{attribute 'qualified_only'}
// ------------------------------------------------------------------------- 
//  SRCI Robot Library                                                
// ------------------------------------------------------------------------- 
//                                                                           
//  Object:      TriggerModeLimit                                       
//  Author:      Thorsten Brach                                                
//  Date:        2024-06-01
//
//  Description:                                              
//   
//                                                                           
//  Copyright: 
//    (C) 2024 Thorsten Brach. All rights reserved                                                                         
//                                                                           
//  Disclaimer:                                                                           
//    This project is provided without any guarantee and can be used for   
//    private and commercial purposes. Any commercial use is at the user’s 
//    own risk and responsibility.
//
// -------------------------------------------------------------------------
TYPE TriggerModeLimit :
(
	/// 0: Invalid (default)
  INVALID := 0,
  /// 1: Joint current in mA
  JOINT_CURRENT := 1,
  /// 2: Force in Nm
  FORCE := 2,
  /// 3: Following error. The distance of the robot position from the path that was calculated
  FOLLOWING_ERROR := 3,
  /// Temperature in °C
  TEMPERATURE := 4  
)SINT;
END_TYPE

{attribute 'qualified_only'}
// ------------------------------------------------------------------------- 
//  SRCI Robot Library                                                
// ------------------------------------------------------------------------- 
//                                                                           
//  Object:      TriggerModeMeasurement                                       
//  Author:      Thorsten Brach                                                
//  Date:        2024-06-01
//
//  Description:                                              
//   
//                                                                           
//  Copyright: 
//    (C) 2024 Thorsten Brach. All rights reserved                                                                         
//                                                                           
//  Disclaimer:                                                                           
//    This project is provided without any guarantee and can be used for   
//    private and commercial purposes. Any commercial use is at the user’s 
//    own risk and responsibility.
//
// -------------------------------------------------------------------------
TYPE TriggerModeMeasurement :
(
	/// (default) No trigger related behavior
  NO_TRIGGER := 0,
  /// 1: Starts the measurement with the positive trigger event and stops it with the negative trigger event 
  ///    when the trigger function with the identical EmitterID is activated.
  POSITIVE_START_NEGATIVE_STOP := 1,
  /// 2: Starts and stops the measurement with the positive trigger event 
  ///    when the trigger function with the identical EmitterID is activated.
  POSITIVE_START_STOP := 2
)USINT;
END_TYPE

{attribute 'qualified_only'}
// ------------------------------------------------------------------------- 
//  SRCI Robot Library                                                
// ------------------------------------------------------------------------- 
//                                                                           
//  Object:      TriggerReactionMode                                       
//  Author:      Thorsten Brach                                                
//  Date:        2024-06-01
//
//  Description:                                              
//   
//                                                                           
//  Copyright: 
//    (C) 2024 Thorsten Brach. All rights reserved                                                                         
//                                                                           
//  Disclaimer:                                                                           
//    This project is provided without any guarantee and can be used for   
//    private and commercial purposes. Any commercial use is at the user’s 
//    own risk and responsibility.
//
// -------------------------------------------------------------------------
TYPE TriggerReactionMode :
(
/// No reaction (default).
  NO_REACTION := 0,
  /// Interrupt: Robot movement is paused. Movement can be continued by function GroupContinue.
  INTERRUPT := 1,
  /// GroupStop: Robot stops the movement and brings all axes to a halt. Movements aborted by this command cannot be continued.
  GROUP_STOP := 2,
  /// Disable robot: The robot’s drives are disabled. This leads to the robot state "Not enabled" (see chapter 5.5.3).
  DISABLE_ROBOT := 3,
  /// Stop actual motion command: Robot movement is paused. Movement can be continued by the next motion command.
  STOP_ACTUAL_MOTION_COMMAND := 4
)SINT;
END_TYPE

{attribute 'qualified_only'}
// ------------------------------------------------------------------------- 
//  SRCI Robot Library                                                
// ------------------------------------------------------------------------- 
//                                                                           
//  Object:      TurnMode                                       
//  Author:      Thorsten Brach                                                
//  Date:        2024-06-01
//
//  Description:                                              
//   
//                                                                           
//  Copyright: 
//    (C) 2024 Thorsten Brach. All rights reserved                                                                         
//                                                                           
//  Disclaimer:                                                                           
//    This project is provided without any guarantee and can be used for   
//    private and commercial purposes. Any commercial use is at the user’s 
//    own risk and responsibility.
//
// -------------------------------------------------------------------------
TYPE TurnMode :
(
  /// Use TurnNumber in position
	USE_TURN_NUMBER := 0,
  ///  Do not change TurnNumber with this movement
  SAME            := 1,
  /// TurnNumber in position is not used but the Robot is free to change TurnNumber
  FREE            := 2
)USINT;
END_TYPE

{attribute 'qualified_only'}
// ------------------------------------------------------------------------- 
//  SRCI Robot Library                                                
// ------------------------------------------------------------------------- 
//                                                                           
//  Object:      WorkAreaReactionMode                                       
//  Author:      Thorsten Brach                                                
//  Date:        2024-06-01
//
//  Description:                                              
//   
//                                                                           
//  Copyright: 
//    (C) 2024 Thorsten Brach. All rights reserved                                                                         
//                                                                           
//  Disclaimer:                                                                           
//    This project is provided without any guarantee and can be used for   
//    private and commercial purposes. Any commercial use is at the user’s 
//    own risk and responsibility.
//
// -------------------------------------------------------------------------
TYPE WorkAreaReactionMode :
(
  /// 0: No reaction (default)
  /// • RC reports violation
  /// • Robot is not stopped
  NO_REACTION := 0,
  /// 
  /// 1: Abort
  /// • RC reports violation
  /// • RC returns error
  /// • Robot is stopped
  /// • Sequence buffer emptied
  ABORT := 1,
  /// 2: Interrupt
  /// • RC reports violation
  /// • Robot movement is paused
  /// • Movement can be continued by function GroupContinue
   INTERRUPT := 2
)USINT;
END_TYPE

{attribute 'qualified_only'}
// ------------------------------------------------------------------------- 
//  SRCI Robot Library                                                
// ------------------------------------------------------------------------- 
//                                                                           
//  Object:      ActiveCommandRegisterState                                       
//  Author:      Thorsten Brach                                                
//  Date:        2024-06-01
//
//  Description:                                              
//   
//                                                                           
//  Copyright: 
//    (C) 2024 Thorsten Brach. All rights reserved                                                                         
//                                                                           
//  Disclaimer:                                                                           
//    This project is provided without any guarantee and can be used for   
//    private and commercial purposes. Any commercial use is at the user’s 
//    own risk and responsibility.
//
// -------------------------------------------------------------------------
TYPE ActiveCommandRegisterState :
(
  /// IS_FREE denotes not used but available resources (empty slots in the ACR).
	IS_FREE        := 0,
  /// IS_PROCESSING CMDs are actively being processed by client or server. 
  /// In terms of CMD category, IS_PROCESSING also describes commands whose tasks are not currently being executed (not ACTIVE), 
  /// but e.g. a CMD waiting in the Sequence buffer.
  IS_PROCESSING := 1,
  /// IS_FINAL states are reached on CMD termination. Execution of this Task has been finished and its results can be examined.
  IS_FINAL    := 2
);
END_TYPE

{attribute 'qualified_only'}
// ------------------------------------------------------------------------- 
//  SRCI Robot Library                                                
// ------------------------------------------------------------------------- 
//                                                                           
//  Object:      BufferStateCmd                                       
//  Author:      Thorsten Brach                                                
//  Date:        2024-06-01
//
//  Description:                                              
//   
//                                                                           
//  Copyright: 
//    (C) 2024 Thorsten Brach. All rights reserved                                                                         
//                                                                           
//  Disclaimer:                                                                           
//    This project is provided without any guarantee and can be used for   
//    private and commercial purposes. Any commercial use is at the user’s 
//    own risk and responsibility.
//
// -------------------------------------------------------------------------
TYPE BufferStateCmd :
(
 // PDF Seite 353 
  EMPTY            := 0,
	CREATED          := 1,
  UPDATE_AVAILABLE := 2,
  SENDING          := 3,
  PROCESSED        := 4  
);
END_TYPE

{attribute 'qualified_only'}
// ------------------------------------------------------------------------- 
//  SRCI Robot Library                                                
// ------------------------------------------------------------------------- 
//                                                                           
//  Object:      BufferStateRsp                                       
//  Author:      Thorsten Brach                                                
//  Date:        2024-06-01
//
//  Description:                                              
//   
//                                                                           
//  Copyright: 
//    (C) 2024 Thorsten Brach. All rights reserved                                                                         
//                                                                           
//  Disclaimer:                                                                           
//    This project is provided without any guarantee and can be used for   
//    private and commercial purposes. Any commercial use is at the user’s 
//    own risk and responsibility.
//
// -------------------------------------------------------------------------
TYPE BufferStateRsp :
(
 // PDF Seite 353 
  EMPTY            := 0,
  RECEIVING        := 1,
  RECEIVED         := 2,
  PROCESSED        := 3  
);
END_TYPE

{attribute 'qualified_only'}
// ------------------------------------------------------------------------- 
//  SRCI Robot Library                                                
// ------------------------------------------------------------------------- 
//                                                                           
//  Object:      CmdMessageState                                       
//  Author:      Thorsten Brach                                                
//  Date:        2024-06-01
//
//  Description:                                              
//   
//                                                                           
//  Copyright: 
//    (C) 2024 Thorsten Brach. All rights reserved                                                                         
//                                                                           
//  Disclaimer:                                                                           
//    This project is provided without any guarantee and can be used for   
//    private and commercial purposes. Any commercial use is at the user’s 
//    own risk and responsibility.
//
// -------------------------------------------------------------------------
TYPE CmdMessageState :
(
  /// No operation or process is active
  EMPTY := 0,
  /// Created but not yet started
  CREATED := 1,
  /// Buffered and awaiting execution
  BUFFERED := 2,
  /// Buffered in planner for future execution
  BUFFERED_IN_PLANNER := 3,
  /// Currently active and in progress
  ACTIVE := 4,
  /// Interrupted and awaiting continuation
  INTERRUPTED := 5,
  /// Requested for abort
  ABORT_REQUEST := 6,
  /// Successfully completed
  DONE := 10,
  /// Aborted before completion
  ABORTED := 14,
  /// Encountered an error during execution
  ERROR := 15
)USINT;
END_TYPE

{attribute 'qualified_only'}
// ------------------------------------------------------------------------- 
//  SRCI Robot Library                                                
// ------------------------------------------------------------------------- 
//                                                                           
//  Object:      InitializationState                                       
//  Author:      Thorsten Brach                                                
//  Date:        2024-06-01
//
//  Description:                                              
//   
//                                                                           
//  Copyright: 
//    (C) 2024 Thorsten Brach. All rights reserved                                                                         
//                                                                           
//  Disclaimer:                                                                           
//    This project is provided without any guarantee and can be used for   
//    private and commercial purposes. Any commercial use is at the user’s 
//    own risk and responsibility.
//
// -------------------------------------------------------------------------
TYPE InitializationState :
(
  /// Default
  DEFAULT := 0,
  /// Error: Telegram control does not match the telegram state
  ERROR_TELEGRAM_CONTROL := 161,
  /// Error: Initialization lost for unknown reason. See message log after reinitializing
  ERROR_INIT_LOST := 162,
  /// Error: Telegram length does not match the length provided in the communication interface.
  ERROR_TELEGRAM_LENGTH := 163,
  /// Error: Incompatible major SRCI version
  ERROR_INCOMPATIBLE_SRCI := 164,
  /// Error: Lifesign timeout
  ERROR_LIFESIGN_TIMEOUT := 165,
  /// Error: The selected optional cyclic data does not fit in the given telegram size
  ERROR_CYCLIC_DATA_MISMATCH := 166,
  /// Error: The robot interface was reset after being initialized
  ERROR_INTERFACE_RESET := 167,
  /// Error: Telegram sequence timeout
  ERROR_SEQUENCE_TIMEOUT := 168,
  /// Error: The telegram number changed after initialization
  ERROR_TELEGRAM_NUMBER_CHANGED := 169,
  /// Error: Invalid AxesGroupID
  ERROR_INVALID_AXES_GROUP := 170,
  /// Error: Telegram number is invalid. E.g. TwoSequences is only activated in one direction
  ERROR_INVALID_TELEGRAM_NUMBER := 171,
  /// Error: Telegram Number is not supported
  ERROR_TELEGRAM_NUMBER_NOT_SUPPORTED := 172,
  /// Ready to resume: The RC is currently not initialized but has state in the ACR
  READY_TO_RESUME := 253,
  /// Ready for initialization: The RC is currently not initialized and has no state in the ACR
  READY_FOR_INITIALIZATION := 254,
  /// Initialized: The RC state is Initialized
  INITIALIZED := 255
);
END_TYPE

{attribute 'qualified_only'}
// ------------------------------------------------------------------------- 
//  SRCI Robot Library                                                
// ------------------------------------------------------------------------- 
//                                                                           
//  Object:      RaPowerState                                       
//  Author:      Thorsten Brach                                                
//  Date:        2024-06-01
//
//  Description:                                              
//   
//                                                                           
//  Copyright: 
//    (C) 2024 Thorsten Brach. All rights reserved                                                                         
//                                                                           
//  Disclaimer:                                                                           
//    This project is provided without any guarantee and can be used for   
//    private and commercial purposes. Any commercial use is at the user’s 
//    own risk and responsibility.
//
// -------------------------------------------------------------------------
TYPE RaPowerState :
(
  /// Robot drives disabled. Robot cannot be moved
	NOT_ENABLED := 0,
  /// Robot drives powered on. Robot can be moved according to sequence state
  ENABLED := 1
)USINT;
END_TYPE

{attribute 'qualified_only'}
// ------------------------------------------------------------------------- 
//  SRCI Robot Library                                                
// ------------------------------------------------------------------------- 
//                                                                           
//  Object:      RaSequenceState                                       
//  Author:      Thorsten Brach                                                
//  Date:        2024-06-01
//
//  Description:                                              
//   
//                                                                           
//  Copyright: 
//    (C) 2024 Thorsten Brach. All rights reserved                                                                         
//                                                                           
//  Disclaimer:                                                                           
//    This project is provided without any guarantee and can be used for   
//    private and commercial purposes. Any commercial use is at the user’s 
//    own risk and responsibility.
//
// -------------------------------------------------------------------------
TYPE RaSequenceState :
(
  /// Robot can be moved by incoming command
	IDLE := 0,
  /// RC is processing command in active sequence
  EXECUTING := 1,
  /// Interrupt is active. Robot is waiting for Continue
  INTERRUPTED := 2
)USINT;
END_TYPE

{attribute 'qualified_only'}
// ------------------------------------------------------------------------- 
//  SRCI Robot Library                                                
// ------------------------------------------------------------------------- 
//                                                                           
//  Object:      RiState                                       
//  Author:      Thorsten Brach                                                
//  Date:        2024-06-01
//
//  Description:                                              
//   
//                                                                           
//  Copyright: 
//    (C) 2024 Thorsten Brach. All rights reserved                                                                         
//                                                                           
//  Disclaimer:                                                                           
//    This project is provided without any guarantee and can be used for   
//    private and commercial purposes. Any commercial use is at the user’s 
//    own risk and responsibility.
//
// -------------------------------------------------------------------------
TYPE RiState :
(
  /// RI is not initialized
	NOT_INITIALIZED := 0,
  /// Initialization finished successfully
  INITIALIZED := 1,
  /// Data between RC and PLC has been synchronized
  SYNCHRONIZED := 2
)USINT;
END_TYPE

{attribute 'qualified_only'}
// ------------------------------------------------------------------------- 
//  SRCI Robot Library                                                
// ------------------------------------------------------------------------- 
//                                                                           
//  Object:      AreaType                                       
//  Author:      Thorsten Brach                                                
//  Date:        2024-06-01
//
//  Description:                                              
//   
//                                                                           
//  Copyright: 
//    (C) 2024 Thorsten Brach. All rights reserved                                                                         
//                                                                           
//  Disclaimer:                                                                           
//    This project is provided without any guarantee and can be used for   
//    private and commercial purposes. Any commercial use is at the user’s 
//    own risk and responsibility.
//
// -------------------------------------------------------------------------
TYPE AreaType :
(
  /// 0: Axes
	AXES := 0,
  /// 1: Box (default)
  BOX := 1,
  /// 2: Cylinder
  CYLINDER := 2,
  /// 3: Sphere (only DefinitionMode 1)
  SPHERE := 3
)USINT;
END_TYPE

{attribute 'qualified_only'}
// ------------------------------------------------------------------------- 
//  SRCI Robot Library                                                
// ------------------------------------------------------------------------- 
//                                                                           
//  Object:      AxesGroupParameterCmdEntries                                       
//  Author:      Thorsten Brach                                                
//  Date:        2024-06-01
//
//  Description:                                              
//   
//                                                                           
//  Copyright: 
//    (C) 2024 Thorsten Brach. All rights reserved                                                                         
//                                                                           
//  Disclaimer:                                                                           
//    This project is provided without any guarantee and can be used for   
//    private and commercial purposes. Any commercial use is at the user’s 
//    own risk and responsibility.
//
// -------------------------------------------------------------------------
TYPE AxesGroupParameterCmdEntries :
(
  /// Handles multiple mechanisms required for operation of the interface
  RobotTask := 0, // No function code  
  /// Read robot-specific data from the RC
  ReadRobotData := 9002,  
  /// Enable/Disable robot into RA power state "Enabled"
  EnableRobot := 1,  
  /// Acknowledgement all pending errors
  GroupReset := 2,  
  /// Read the actual position – TCP: X…RZ + config/Turn, Joint: (J1…E6)
  ReadActualPosition := 3,
  /// Read the actual position cyclically
  ReadActualPositionCyclic := 4,   
  /// Read D-H-parameters of robot
  ReadDHParameter := 5,  
  /// Restart/reboot of the RC
  RestartController := 6,  
  /// Read actual TCP velocity
  ReadActualTCPVelocity := 7,  
  /// Login on RC from PLC
  UserLogin := 8,  
  /// Switch language of robot teach pendant from PLC
  SwitchLanguage := 9,  
  /// Reads and writes specific configuration parameters on RC that are required for the RI to work
  ExchangeConfiguration := 10,  
  /// Set active sequence
  SetSequence := 11,  
  /// Change actual speed override
  ChangeSpeedOverride := 12,  
  /// Read error codes of pending errors and move them into user data block "RobotData"
  ReadMessages := 13,  
  /// Read reference values of robot dynamics for path movement
  ReadRobotReferenceDynamics := 14,  
  /// Change configuration of selected user frame number
  WriteFrameData := 15,  
  /// Change configuration of selected tool number
  WriteToolData := 16,  
  /// Change configuration of selected payload number
  WriteLoadData := 17,  
  /// Write reference values of robot dynamics for path movement
  WriteRobotReferenceDynamics := 18,  
  /// Write default values of dynamic parameters used by move commands
  WriteRobotDefaultDynamics := 19,  
  /// Read default values of dynamic parameters used by move commands
  ReadRobotDefaultDynamics := 20,  
  /// Read content of selected user frame number
  ReadFrameData := 21,  
  /// Read content of selected tool number
  ReadToolData := 22,  
  /// Read content of selected payload number
  ReadLoadData := 23,  
  /// Read actual software limits of the axes Positive and negative Limit of Joint J1…J6, E1…E6
  ReadRobotSWLimits := 24,  
  /// Change robot limits of robot axes (degree)
  WriteRobotSWLimits := 25,  
  /// Switch operation mode of RC (Automatic External, T1 External, T2 External)
  SetOperationMode := 26,  
  /// Read configuration of defined work areas
  ReadWorkArea := 27,  
  /// Define work area
  WriteWorkArea := 28,  
  /// Enable/Disable work areas of RC and check if TCP is inside/outside of active work area
  ActivateWorkArea := 29,  
  /// Monitor enabled work areas
  MonitorWorkArea := 30,  
  /// Jog robot manually
  GroupJog := 31,  
  /// Move the TCP to an absolute cartesian position (linear interpolation)
  MoveLinearAbsolute := 32,  
  /// Move Joints to an absolute cartesian position (Absolute cartesian PTP) (Joint interpolated movement)
  MoveDirectAbsolute := 33,  
  /// Move all joints to an absolute joint position (Absolute Joint PTP)
  MoveAxesAbsolute := 34,  
  /// Abort actual movement and delete buffer
  GroupStop := 35,  
  /// Interrupt active movement, possible to continue movement
  GroupInterrupt := 36,  
  /// Continue interrupted path
  GroupContinue := 37,  
  /// Move the TCP relative to the actual cartesian position (linear interpolation)
  MoveLinearRelative := 38,  
  /// Move Joints relative to relative cartesian position (Relative cartesian PTP) (Joint interpolated movement)
  MoveDirectRelative := 39,  
  /// Move all joints relative to actual joint position (Relative Joint PTP)
  MoveAxesRelative := 40,  
  /// Return to path left during active interrupt
  ReturnToPrimary := 41,  
  /// Move the TCP to an absolute joint position (linear interpolation)
  MoveCircularAbsolute := 42,  
  /// Move the TCP relative to the actual cartesian position (circular interpolation)
  MoveCircularRelative := 43,  
  /// Move the TCP relative to a reference cartesian position (linear interpolation)
  MoveLinearOffset := 44,  
  /// Move the TCP relative to a reference cartesian position (PTPT interpolation)
  MoveDirectOffset := 45,  
  /// Set wait command between motion commands
  WaitTime := 46,  
  /// Linear Move to target position through auxiliary position defined by offset in all dimensions (movement to target position linear)
  MoveApproachLinear := 47,  
  /// Linear Move from actual position to destination through auxiliary position defined by offset in all dimensions (movement to target position linear)
  MoveDepartLinear := 48,  
  /// Direct Move to target position through auxiliary position defined by offset in all dimensions (movement to target posi tion PTP)
  MoveApproachDirect := 49,  
  /// Direct Move from actual position to destination through auxiliary position defined by offset in all dimensions (movement to the target position PTP)
  MoveDepartDirect := 50,  
  /// Move robot into contact with obstruction (mechanical Limit) and hold it in this position
  SearchHardstop := 51,  
  /// Move robot into contact with obstruction (mechanical Limit) and hold it in this position
  SearchHardstopJ := 52,  
  /// Command several interpolated movement of robot arm on linear paths from actual position
  MovePickPlaceLinear := 53,  
  /// Commands interpolated movement of robot arm on a partly undefined path from actual position
  MovePickPlaceDirect := 54,  
  /// Activate conveyor tracking mode
  ActivateConveyorTracking := 55,  
  /// Redefine tracking position for conveyor tracking
  RedefineTrackingPos := 56,  
  /// Synchronize robot with conveyor
  SyncToConveyor := 57,  
  /// Configure conveyor parameters
  ConfigureConveyor := 58,  
  /// Activate superimposed motion of TCP to defined motion
  MoveSuperImposed := 59,  
  /// Activate superimposed motion of TCP to defined motion
  MoveSuperImposedDynamic := 60,  
  /// Read digital input and output group of RC
  ReadDigitalInputs := 61,  
  /// Read digital output group of RC
  ReadDigitalOutputs := 62,  
  /// Write digital output group of RC
  WriteDigitalOutputs := 63,  
  /// Read integer values on RC
  ReadIntegers := 64,  
  /// Read real values on RC
  ReadReals := 65,  
  /// Write integer values on RC
  WriteIntegers := 66,  
  /// Write real values on RC
  WriteReals := 67,  
  /// Set trigger in defined position of path (L = Linear Path) (cartesian) switch periphery.
  MoveLinearCam := 68,  
  /// Set a trigger in a defined position of a path. (PTP)
  MoveDirectCam := 69,  
  /// Set a trigger in a defined position of a circular path
  MoveCircularCam := 70,  
  /// Read analog input of RC
  ReadAnalogInput := 71,  
  /// Read analog output of RC
  ReadAnalogOutput := 72,  
  /// Write analog output of RC
  WriteAnalogOutput := 73,  
  /// Capture trigger Position, measuring input
  MeasuringInput := 74,  
  /// Abort triggering of Position, measuring input
  AbortMeasuringInput := 75,  
  /// Trigger "Actions" based on I/O related events (e.g. change of DI’s state)
  SetTriggerRegister := 76,  
  /// Trigger "Actions" based on physical events (e.g. force limit reached)
  SetTriggerLimit := 77,  
  /// Trigger "Actions" based on physical events (e.g. force limit reached)
  SetTriggerUser := 78,  
  /// Trigger "Actions" based on incoming error event
  SetTriggerError := 79,  
  /// "Action" that initiates specified events when triggered
  ReactAtTrigger := 80,  
  /// Wait to process next command in sequence until trigger signal is received
  WaitForTrigger := 81,  
  /// Read specific parameter of the robot
  ReadSystemVariable := 82,  
  /// Change value of specific vendor parameter
  WriteSystemVariable := 83,  
  /// Calculate Forward Kinematic
  CalculateForwardKinematic := 84,  
  /// Calculate Inverse Kinematic
  CalculateInverseKinematic := 85,  
  /// Calculate cartesian position from existing cartesian position
  CalculateCartesianPosition := 86,  
  /// Calculate tool (TCP) with four-point method
  CalculateTool := 87,  
  /// Calculate frame with three-point method
  CalculateFrame := 88,  
  /// Cancel currently active move command and continue with the next buffered command
  ActivateNextCommand := 89,  
  /// Transform a defined position in space
  ShiftPosition := 90,  
  /// Trigger an action based on a motion-related parameter (e.g. progress of trajectory)
  SetTriggerMotion := 91,  
  /// Release robot arm’s brakes
  OpenBrake := 92,  
  /// Call subprogram stored in RC from PLC
  CallSubprogram := 93,  
  /// Writes cyclic data of called subprogram
  WriteCallSubprogramCyclic := 94,
  /// Reads cyclic data of called subprogram
  ReadCallSubprogramCyclic := 95,
  /// Stops an active subprogram
  StopSubprogram := 96,  
  /// Switch path mode between high and low accuracy
  PathAccuracyMode := 97,  
  /// Activate/Deactivate functionality to avoid singularities
  AvoidSingularity := 98,  
  /// Enables the RC to apply user-defined force/torque through RA’s TCP movement
  ForceControl := 99,  
  /// Commands specified reaction from RA when defined force/torque detected
  ForceLimit := 100,  
  /// Read actual force/torque at TCP
  ReadActualForce := 101,  
  /// Activate robot cycle brake test and give feedback to PLC
  BrakeTest := 102,  
  /// Push robot: Robot calculates opposite vector and moves slowly in that direction
  SoftSwitchTCP := 103,  
  /// Create spline on RC from positions stored in PLC
  CreateSpline := 104,  
  /// Delete spline previously created on RC
  DeleteSpline := 105,  
  /// Move spline previously created on RC
  MoveSpline := 106,  
  /// Create and move spline on RC simultaneously
  DynamicSpline := 107,  
  /// Automatic detection of load data
  LoadMeasurementAutomatic := 108,  
  /// Sequential detection of load data
  LoadMeasurementSequential := 109,  
  /// Turn on/off the collision detection
  CollisionDetection := 110,  
  /// Move the robot axes by hand
  FreeDrive := 111,  
  /// Measure the length of objects in the cartesian space, execution time for specified section of a job or signal output time of a specified signal
  UnitMeasurement := 112,
  /// Maximum entry
  MAX_ENTRY := 113   
)UINT;
END_TYPE

{attribute 'qualified_only'}
// ------------------------------------------------------------------------- 
//  SRCI Robot Library                                                
// ------------------------------------------------------------------------- 
//                                                                           
//  Object:      CmdType                                       
//  Author:      Thorsten Brach                                                
//  Date:        2024-06-01
//
//  Description:                                              
//   
//                                                                           
//  Copyright: 
//    (C) 2024 Thorsten Brach. All rights reserved                                                                         
//                                                                           
//  Disclaimer:                                                                           
//    This project is provided without any guarantee and can be used for   
//    private and commercial purposes. Any commercial use is at the user’s 
//    own risk and responsibility.
//
// -------------------------------------------------------------------------
TYPE CmdType :
(
  /// Handles multiple mechanisms required for operation of the interface
  RobotTask := 0, // No function code  
  /// Read robot-specific data from the RC
  ReadRobotData := 9002,  
  /// Enable/Disable robot into RA power state "Enabled"
  EnableRobot := 1000,  
  /// Acknowledgement all pending errors
  GroupReset := 1001,  
  /// Read the actual position – TCP: X…RZ + config/Turn, Joint: (J1…E6)
  ReadActualPosition := 5100,
  /// Read the actual position cyclically
  ReadActualPositionCyclic := 1, // No function code  
  /// Read D-H-parameters of robot
  ReadDHParameter := 5101,  
  /// Restart/reboot of the RC
  RestartController := 1101,  
  /// Read actual TCP velocity
  ReadActualTCPVelocity := 5111,  
  /// Login on RC from PLC
  UserLogin := 1006,  
  /// Switch language of robot teach pendant from PLC
  SwitchLanguage := 1005,  
  /// Reads and writes specific configuration parameters on RC that are required for the RI to work
  ExchangeConfiguration := 9000,  
  /// Set active sequence
  SetSequence := 1004,  
  /// Change actual speed override
  ChangeSpeedOverride := 2000,  
  /// Read error codes of pending errors and move them into user data block "RobotData"
  ReadMessages := 9001,  
  /// Read reference values of robot dynamics for path movement
  ReadRobotReferenceDynamics := 5105,  
  /// Change configuration of selected user frame number
  WriteFrameData := 5200,  
  /// Change configuration of selected tool number
  WriteToolData := 5205,  
  /// Change configuration of selected payload number
  WriteLoadData := 5201,  
  /// Write reference values of robot dynamics for path movement
  WriteRobotReferenceDynamics := 5203,  
  /// Write default values of dynamic parameters used by move commands
  WriteRobotDefaultDynamics := 5202,  
  /// Read default values of dynamic parameters used by move commands
  ReadRobotDefaultDynamics := 5104,  
  /// Read content of selected user frame number
  ReadFrameData := 5102,  
  /// Read content of selected tool number
  ReadToolData := 5107,  
  /// Read content of selected payload number
  ReadLoadData := 5103,  
  /// Read actual software limits of the axes Positive and negative Limit of Joint J1…J6, E1…E6
  ReadRobotSWLimits := 5106,  
  /// Change robot limits of robot axes (degree)
  WriteRobotSWLimits := 5204,  
  /// Switch operation mode of RC (Automatic External, T1 External, T2 External)
  SetOperationMode := 1003,  
  /// Read configuration of defined work areas
  ReadWorkArea := 7502,  
  /// Define work area
  WriteWorkArea := 7503,  
  /// Enable/Disable work areas of RC and check if TCP is inside/outside of active work area
  ActivateWorkArea := 7500,  
  /// Monitor enabled work areas
  MonitorWorkArea := 7501,  
  /// Jog robot manually
  GroupJog := 2100,  
  /// Move the TCP to an absolute cartesian position (linear interpolation)
  MoveLinearAbsolute := 2103,  
  /// Move Joints to an absolute cartesian position (Absolute cartesian PTP) (Joint interpolated movement)
  MoveDirectAbsolute := 2102,  
  /// Move all joints to an absolute joint position (Absolute Joint PTP)
  MoveAxesAbsolute := 2101,  
  /// Abort actual movement and delete buffer
  GroupStop := 2003,  
  /// Interrupt active movement, possible to continue movement
  GroupInterrupt := 2002,  
  /// Continue interrupted path
  GroupContinue := 2001,  
  /// Move the TCP relative to the actual cartesian position (linear interpolation)
  MoveLinearRelative := 2110,  
  /// Move Joints relative to relative cartesian position (Relative cartesian PTP) (Joint interpolated movement)
  MoveDirectRelative := 2108,  
  /// Move all joints relative to actual joint position (Relative Joint PTP)
  MoveAxesRelative := 2105,  
  /// Return to path left during active interrupt
  ReturnToPrimary := 2104,  
  /// Move the TCP to an absolute joint position (linear interpolation)
  MoveCircularAbsolute := 2109,  
  /// Move the TCP relative to the actual cartesian position (circular interpolation)
  MoveCircularRelative := 2106,  
  /// Move the TCP relative to a reference cartesian position (linear interpolation)
  MoveLinearOffset := 2112,  
  /// Move the TCP relative to a reference cartesian position (PTPT interpolation)
  MoveDirectOffset := 2111,  
  /// Set wait command between motion commands
  WaitTime := 7005,  
  /// Linear Move to target position through auxiliary position defined by offset in all dimensions (movement to target position linear)
  MoveApproachLinear := 2201,  
  /// Linear Move from actual position to destination through auxiliary position defined by offset in all dimensions (movement to target position linear)
  MoveDepartLinear := 2203,  
  /// Direct Move to target position through auxiliary position defined by offset in all dimensions (movement to target posi tion PTP)
  MoveApproachDirect := 2200,  
  /// Direct Move from actual position to destination through auxiliary position defined by offset in all dimensions (movement to the target position PTP)
  MoveDepartDirect := 2202,  
  /// Move robot into contact with obstruction (mechanical Limit) and hold it in this position
  SearchHardstop := 2500,  
  /// Move robot into contact with obstruction (mechanical Limit) and hold it in this position
  SearchHardstopJ := 2501,  
  /// Command several interpolated movement of robot arm on linear paths from actual position
  MovePickPlaceLinear := 2205,  
  /// Commands interpolated movement of robot arm on a partly undefined path from actual position
  MovePickPlaceDirect := 2204,  
  /// Activate conveyor tracking mode
  ActivateConveyorTracking := 2300,  
  /// Redefine tracking position for conveyor tracking
  RedefineTrackingPos := 2302,  
  /// Synchronize robot with conveyor
  SyncToConveyor := 2303,  
  /// Configure conveyor parameters
  ConfigureConveyor := 2301,  
  /// Activate superimposed motion of TCP to defined motion
  MoveSuperImposed := 2502,  
  /// Activate superimposed motion of TCP to defined motion
  MoveSuperImposedDynamic := 2503,  
  /// Read digital input and output group of RC
  ReadDigitalInputs := 6100,  
  /// Read digital output group of RC
  ReadDigitalOutputs := 6101,  
  /// Write digital output group of RC
  WriteDigitalOutputs := 6104,  
  /// Read integer values on RC
  ReadIntegers := 6102,  
  /// Read real values on RC
  ReadReals := 6103,  
  /// Write integer values on RC
  WriteIntegers := 6105,  
  /// Write real values on RC
  WriteReals := 6106,  
  /// Set trigger in defined position of path (L = Linear Path) (cartesian) switch periphery.
  MoveLinearCam := 2402,  
  /// Set a trigger in a defined position of a path. (PTP)
  MoveDirectCam := 2401,  
  /// Set a trigger in a defined position of a circular path
  MoveCircularCam := 2400,  
  /// Read analog input of RC
  ReadAnalogInput := 6107,  
  /// Read analog output of RC
  ReadAnalogOutput := 6108,  
  /// Write analog output of RC
  WriteAnalogOutput := 6109,  
  /// Capture trigger Position, measuring input
  MeasuringInput := 6001,  
  /// Abort triggering of Position, measuring input
  AbortMeasuringInput := 6000,  
  /// Trigger "Actions" based on I/O related events (e.g. change of DI’s state)
  SetTriggerRegister := 3004,  
  /// Trigger "Actions" based on physical events (e.g. force limit reached)
  SetTriggerLimit := 3002,  
  /// Trigger "Actions" based on physical events (e.g. force limit reached)
  SetTriggerUser := 3005,  
  /// Trigger "Actions" based on incoming error event
  SetTriggerError := 3001,  
  /// "Action" that initiates specified events when triggered
  ReactAtTrigger := 3000,  
  /// Wait to process next command in sequence until trigger signal is received
  WaitForTrigger := 3006,  
  /// Read specific parameter of the robot
  ReadSystemVariable := 5109,  
  /// Change value of specific vendor parameter
  WriteSystemVariable := 5206,  
  /// Calculate Forward Kinematic
  CalculateForwardKinematic := 7203,  
  /// Calculate Inverse Kinematic
  CalculateInverseKinematic := 7204,  
  /// Calculate cartesian position from existing cartesian position
  CalculateCartesianPosition := 7200,  
  /// Calculate tool (TCP) with four-point method
  CalculateTool := 7202,  
  /// Calculate frame with three-point method
  CalculateFrame := 7201,  
  /// Cancel currently active move command and continue with the next buffered command
  ActivateNextCommand := 7000,  
  /// Transform a defined position in space
  ShiftPosition := 7205,  
  /// Trigger an action based on a motion-related parameter (e.g. progress of trajectory)
  SetTriggerMotion := 3003,  
  /// Release robot arm’s brakes
  OpenBrake := 7100,  
  /// Call subprogram stored in RC from PLC
  CallSubprogram := 7001,  
  /// Writes cyclic data of called subprogram
  WriteCallSubprogramCyclic := 2, // No function code
  /// Reads cyclic data of called subprogram
  ReadCallSubprogramCyclic := 3, // No function code
  /// Stops an active subprogram
  StopSubprogram := 7008,  
  /// Switch path mode between high and low accuracy
  PathAccuracyMode := 7401,  
  /// Activate/Deactivate functionality to avoid singularities
  AvoidSingularity := 7400,  
  /// Enables the RC to apply user-defined force/torque through RA’s TCP movement
  ForceControl := 7301,  
  /// Commands specified reaction from RA when defined force/torque detected
  ForceLimit := 7302,  
  /// Read actual force/torque at TCP
  ReadActualForce := 5110,  
  /// Activate robot cycle brake test and give feedback to PLC
  BrakeTest := 7101,  
  /// Push robot: Robot calculates opposite vector and moves slowly in that direction
  SoftSwitchTCP := 7300,  
  /// Create spline on RC from positions stored in PLC
  CreateSpline := 2600,  
  /// Delete spline previously created on RC
  DeleteSpline := 2601,  
  /// Move spline previously created on RC
  MoveSpline := 2603,  
  /// Create and move spline on RC simultaneously
  DynamicSpline := 2602,  
  /// Automatic detection of load data
  LoadMeasurementAutomatic := 7006,  
  /// Sequential detection of load data
  LoadMeasurementSequential := 7007,  
  /// Turn on/off the collision detection
  CollisionDetection := 7003,  
  /// Move the robot axes by hand
  FreeDrive := 7002,  
  /// Measure the length of objects in the cartesian space, execution time for specified section of a job or signal output time of a specified signal
  UnitMeasurement := 7004   
)UINT;
END_TYPE

{attribute 'qualified_only'}
// ------------------------------------------------------------------------- 
//  SRCI Robot Library                                                
// ------------------------------------------------------------------------- 
//                                                                           
//  Object:      ConveyorType                                       
//  Author:      Thorsten Brach                                                
//  Date:        2024-06-01
//
//  Description:                                              
//   
//                                                                           
//  Copyright: 
//    (C) 2024 Thorsten Brach. All rights reserved                                                                         
//                                                                           
//  Disclaimer:                                                                           
//    This project is provided without any guarantee and can be used for   
//    private and commercial purposes. Any commercial use is at the user’s 
//    own risk and responsibility.
//
// -------------------------------------------------------------------------
TYPE ConveyorType :
(
  /// Linear Conveyor Tracking (default)
	LINEAR_CONVEYOR_TRACKING := 0,
  /// Circular Conveyor Tracking
  CIRCULAR_CONVEYOR_TRACKING := 1
)USINT;
END_TYPE

{attribute 'qualified_only'}
// ------------------------------------------------------------------------- 
//  SRCI Robot Library                                                
// ------------------------------------------------------------------------- 
//                                                                           
//  Object:      MessageType                                       
//  Author:      Thorsten Brach                                                
//  Date:        2024-06-01
//
//  Description:                                              
//   
//                                                                           
//  Copyright: 
//    (C) 2024 Thorsten Brach. All rights reserved                                                                         
//                                                                           
//  Disclaimer:                                                                           
//    This project is provided without any guarantee and can be used for   
//    private and commercial purposes. Any commercial use is at the user’s 
//    own risk and responsibility.
//
// -------------------------------------------------------------------------
TYPE MessageType :
(
  /// RI related messages
  RI := 1,
  /// RC related messages
  RC := 2,
  /// RA related messages
  RA := 3, 
  /// Command related messages
  CMD := 4 
)USINT;
END_TYPE

{attribute 'qualified_only'}
// ------------------------------------------------------------------------- 
//  SRCI Robot Library                                                
// ------------------------------------------------------------------------- 
//                                                                           
//  Object:      ReferenceType                                       
//  Author:      Thorsten Brach                                                
//  Date:        2024-06-01
//
//  Description:                                              
//   
//                                                                           
//  Copyright: 
//    (C) 2024 Thorsten Brach. All rights reserved                                                                         
//                                                                           
//  Disclaimer:                                                                           
//    This project is provided without any guarantee and can be used for   
//    private and commercial purposes. Any commercial use is at the user’s 
//    own risk and responsibility.
//
// -------------------------------------------------------------------------
TYPE ReferenceType :
(
  /// Distance is applied in the Tool coordinate system. 
  /// The setting of the parameter FrameNo will be ignored.
	TOOL  := 0,
  /// Distance is applied in the Frame coordinate system.
  /// The settings of the ToolNo are also effective and must be considered. 
  FRAME := 1
)USINT;
END_TYPE

{attribute 'qualified_only'}
// ------------------------------------------------------------------------- 
//  SRCI Robot Library                                                
// ------------------------------------------------------------------------- 
//                                                                           
//  Object:      UnitType                                       
//  Author:      Thorsten Brach                                                
//  Date:        2024-06-01
//
//  Description:                                              
//   
//                                                                           
//  Copyright: 
//    (C) 2024 Thorsten Brach. All rights reserved                                                                         
//                                                                           
//  Disclaimer:                                                                           
//    This project is provided without any guarantee and can be used for   
//    private and commercial purposes. Any commercial use is at the user’s 
//    own risk and responsibility.
//
// -------------------------------------------------------------------------
TYPE UnitType :
(
  /// Volt
	VOLT   := 0,
  /// Ampere
  AMPERE := 1
)USINT;
END_TYPE

{attribute 'pack_mode' := '1'} 
// ------------------------------------------------------------------------- 
//  SRCI Robot Library                                                
// ------------------------------------------------------------------------- 
//                                                                           
//  Object:      AxesGroup                                       
//  Author:      Thorsten Brach                                                
//  Date:        2024-06-01
//
//  Description:                                              
//   
//                                                                           
//  Copyright: 
//    (C) 2024 Thorsten Brach. All rights reserved                                                                         
//                                                                           
//  Disclaimer:                                                                           
//    This project is provided without any guarantee and can be used for   
//    private and commercial purposes. Any commercial use is at the user’s 
//    own risk and responsibility.
//
// -------------------------------------------------------------------------
TYPE AxesGroup :
STRUCT
  /// Parameter 
  Parameter      : AxesGroupParameter;
  /// RI state information (see chapter 5.5.3) 
  State          : AxesGroupState;
  /// RC, RA, RI, and CMD warnings and errors (see chapter 5.5.11)
  MessageLog     : AxesGroupMessageLog;
  /// Cyclic data exchanged between server and client (see chapter 5.6.6.5) 
  Cyclic         : AxesGroupCyclic;
  /// Optional cyclic data exchanged between server and client (see chapter 5.6.6.2)
  OptionalCyclic : AxesGroupCyclicOptionalData;
  /// Execution order list and ACR entries (see chapter 5.6.4.2) 
  Acyclic        : AxesGroupAcyclic;
  /// Telegram data (see chapter 5.6.6.2) 
  Config         : Telegram; 
END_STRUCT
END_TYPE

{attribute 'pack_mode' := '1'} 
// ------------------------------------------------------------------------- 
//  SRCI Robot Library                                                
// ------------------------------------------------------------------------- 
//                                                                           
//  Object:      RobotCartesianForce                                       
//  Author:      Thorsten Brach                                                
//  Date:        2024-06-01
//
//  Description:                                              
//   
//                                                                           
//  Copyright: 
//    (C) 2024 Thorsten Brach. All rights reserved                                                                         
//                                                                           
//  Disclaimer:                                                                           
//    This project is provided without any guarantee and can be used for   
//    private and commercial purposes. Any commercial use is at the user’s 
//    own risk and responsibility.
//
// -------------------------------------------------------------------------
TYPE RobotCartesianForce :
STRUCT
  /// Force on the X-Axis
  X : REAL;
  /// Force on the Y-Axis
  Y : REAL;
  /// Force on the Z-Axis
  Z : REAL;
  /// Force around the X-Axis (RX)
  Rx : REAL;
  /// Force around the Y-Axis (RY)
  Ry : REAL;
  /// Force around the Z-Axis (RZ)
  Rz : REAL;
  /// Force of first external axis
  E1 : REAL;
  /// Force of second external axis
  E2 : REAL;
  /// Force of third external axis
  E3 : REAL;
  /// Force of fourth external axis
  E4 : REAL;
  /// Force of fifth external axis
  E5 : REAL;
  /// Force of sixth external axis
  E6 : REAL;    
END_STRUCT
END_TYPE

{attribute 'pack_mode' := '1'} 
// ------------------------------------------------------------------------- 
//  SRCI Robot Library                                                
// ------------------------------------------------------------------------- 
//                                                                           
//  Object:      RobotCartesianForceExt                                       
//  Author:      Thorsten Brach                                                
//  Date:        2024-06-01
//
//  Description:                                              
//   
//                                                                           
//  Copyright: 
//    (C) 2024 Thorsten Brach. All rights reserved                                                                         
//                                                                           
//  Disclaimer:                                                                           
//    This project is provided without any guarantee and can be used for   
//    private and commercial purposes. Any commercial use is at the user’s 
//    own risk and responsibility.
//
// -------------------------------------------------------------------------
TYPE RobotCartesianForceExt :
STRUCT
  /// Force on the first external axis
  E1 : REAL;
  /// Force of second external axis
  E2 : REAL;
  /// Force of third external axis
  E3 : REAL;
  /// Force of fourth external axis
  E4 : REAL;
  /// Force of fifth external axis
  E5 : REAL;
  /// Force of sixth external axis
  E6 : REAL;  
END_STRUCT
END_TYPE

{attribute 'pack_mode' := '1'} 
// ------------------------------------------------------------------------- 
//  SRCI Robot Library                                                
// ------------------------------------------------------------------------- 
//                                                                           
//  Object:      RobotCartesianForceShort                                       
//  Author:      Thorsten Brach                                                
//  Date:        2024-06-01
//
//  Description:                                              
//   
//                                                                           
//  Copyright: 
//    (C) 2024 Thorsten Brach. All rights reserved                                                                         
//                                                                           
//  Disclaimer:                                                                           
//    This project is provided without any guarantee and can be used for   
//    private and commercial purposes. Any commercial use is at the user’s 
//    own risk and responsibility.
//
// -------------------------------------------------------------------------
TYPE RobotCartesianForceShort :
STRUCT
  /// Force on the X-Axis
  X : REAL;
  /// Force on the Y-Axis
  Y : REAL;
  /// Force on the Z-Axis
  Z : REAL;
  /// Force around the X-Axis (RX)
  Rx : REAL;
  /// Force around the Y-Axis (RY)
  Ry : REAL;
  /// Force around the Z-Axis (RZ)
  Rz : REAL;
END_STRUCT
END_TYPE

{attribute 'pack_mode' := '1'} 
// ------------------------------------------------------------------------- 
//  SRCI Robot Library                                                
// ------------------------------------------------------------------------- 
//                                                                           
//  Object:      RobotCartesianPosition                                       
//  Author:      Thorsten Brach                                                
//  Date:        2024-06-01
//
//  Description:                                              
//   
//                                                                           
//  Copyright: 
//    (C) 2024 Thorsten Brach. All rights reserved                                                                         
//                                                                           
//  Disclaimer:                                                                           
//    This project is provided without any guarantee and can be used for   
//    private and commercial purposes. Any commercial use is at the user’s 
//    own risk and responsibility.
//
// -------------------------------------------------------------------------
TYPE RobotCartesianPosition :
STRUCT
  /// TCP Position on the X-Axis
  X          : REAL;
  /// TCP Position on the Y-Axis
  Y          : REAL;
  /// TCP Position on the Z-Axis
  Z          : REAL;
  /// Rotation around the X-Axis (RX)
  Rx         : REAL;
  /// Rotation around the Y-Axis (RY)
  Ry         : REAL;
  /// Rotation around the Z-Axis (RZ)
  Rz         : REAL;
  /// Configuration data of the robot (Config)
  Config     : ArmConfigParameter;
  /// Turn number of the axes (TurnNumber)
  TurnNumber : TurnNumber;
  /// Position of first external axis
  E1         : REAL;  
  /// Position of second external axis
  E2         : REAL;
  /// Position of third external axis
  E3         : REAL;
  /// Position of fourth external axis
  E4         : REAL;
  /// Position of fifth external axis
  E5         : REAL;
  /// Position of sixth external axis
  E6         : REAL;    
END_STRUCT
END_TYPE

{attribute 'pack_mode' := '1'} 
// ------------------------------------------------------------------------- 
//  SRCI Robot Library                                                
// ------------------------------------------------------------------------- 
//                                                                           
//  Object:      RobotCartesianPositionExt                                       
//  Author:      Thorsten Brach                                                
//  Date:        2024-06-01
//
//  Description:                                              
//   
//                                                                           
//  Copyright: 
//    (C) 2024 Thorsten Brach. All rights reserved                                                                         
//                                                                           
//  Disclaimer:                                                                           
//    This project is provided without any guarantee and can be used for   
//    private and commercial purposes. Any commercial use is at the user’s 
//    own risk and responsibility.
//
// -------------------------------------------------------------------------
TYPE RobotCartesianPositionExt :
STRUCT
  /// Position of second external axis
  E2 : REAL;
  /// Position of third external axis
  E3 : REAL;
  /// Position of fourth external axis
  E4 : REAL;
  /// Position of fifth external axis
  E5 : REAL;
  /// Position of sixth external axis
  E6 : REAL;  
END_STRUCT
END_TYPE

{attribute 'pack_mode' := '1'} 
// ------------------------------------------------------------------------- 
//  SRCI Robot Library                                                
// ------------------------------------------------------------------------- 
//                                                                           
//  Object:      RobotCartesianPositionShort                                       
//  Author:      Thorsten Brach                                                
//  Date:        2024-06-01
//
//  Description:                                              
//   
//                                                                           
//  Copyright: 
//    (C) 2024 Thorsten Brach. All rights reserved                                                                         
//                                                                           
//  Disclaimer:                                                                           
//    This project is provided without any guarantee and can be used for   
//    private and commercial purposes. Any commercial use is at the user’s 
//    own risk and responsibility.
//
// -------------------------------------------------------------------------
TYPE RobotCartesianPositionShort :
STRUCT
  /// TCP Position on the X-Axis
  X          : REAL;
  /// TCP Position on the Y-Axis
  Y          : REAL;
  /// TCP Position on the Z-Axis
  Z          : REAL;
  /// Rotation around the X-Axis (RX)
  Rx         : REAL;
  /// Rotation around the Y-Axis (RY)
  Ry         : REAL;
  /// Rotation around the Z-Axis (RZ)
  Rz         : REAL;
  /// Configuration data of the robot (Config)
  Config     : ArmConfigParameter;
  /// Turn number of the axes (TurnNumber)
  TurnNumber : TurnNumber;
  /// Position of first external axis
  E1         : REAL;
END_STRUCT
END_TYPE

{attribute 'pack_mode' := '1'}
// ------------------------------------------------------------------------- 
//  SRCI Robot Library                                                
// ------------------------------------------------------------------------- 
//                                                                           
//  Object:      CmdHeader                                       
//  Author:      Thorsten Brach                                                
//  Date:        2024-06-01
//
//  Description:                                              
//   
//                                                                           
//  Copyright: 
//    (C) 2024 Thorsten Brach. All rights reserved                                                                         
//                                                                           
//  Disclaimer:                                                                           
//    This project is provided without any guarantee and can be used for   
//    private and commercial purposes. Any commercial use is at the user’s 
//    own risk and responsibility.
//
// ------------------------------------------------------------------------- 
TYPE CmdHeader :
STRUCT
  /// Type of command - For more information see chapter 5.6.4.
 CmdTyp          : CmdType;
 /// Specifies target buffer and processing behavior - For more information see chapter 5.6.4.5
 ExecMode        : ExecutionMode;
 /// Parameter Sequence, used to identify sets of CMD parameter
 ParSeq          : SequenceFlag;
 /// Priority of this command
 Priority        : PriorityLevel;  
END_STRUCT
END_TYPE

{attribute 'pack_mode' := '1'} 
// ------------------------------------------------------------------------- 
//  SRCI Robot Library                                                
// ------------------------------------------------------------------------- 
//                                                                           
//  Object:      LogParameter                                       
//  Author:      Thorsten Brach                                                
//  Date:        2024-06-01
//
//  Description:                                              
//   
//                                                                           
//  Copyright: 
//    (C) 2024 Thorsten Brach. All rights reserved                                                                         
//                                                                           
//  Disclaimer:                                                                           
//    This project is provided without any guarantee and can be used for   
//    private and commercial purposes. Any commercial use is at the user’s 
//    own risk and responsibility.
//
// -------------------------------------------------------------------------
TYPE LogParameter :
STRUCT
  /// Log level setting for creating commands  
  CreateCmd : LogLevel;
  /// Log level setting for updating commands
  UpdateCmd : LogLevel;
  /// Log level setting for generating sequence 
  GenSeq    : LogLevel;
  /// Log level for ??? sequence
  DecSeq    : LogLevel;
END_STRUCT
END_TYPE

{attribute 'pack_mode' := '1'} 
// ------------------------------------------------------------------------- 
//  SRCI Robot Library                                                
// ------------------------------------------------------------------------- 
//                                                                           
//  Object:      RobotCoordinateSystemParameters                                       
//  Author:      Thorsten Brach                                                
//  Date:        2024-06-01
//
//  Description:                                              
//   
//                                                                           
//  Copyright: 
//    (C) 2024 Thorsten Brach. All rights reserved                                                                         
//                                                                           
//  Disclaimer:                                                                           
//    This project is provided without any guarantee and can be used for   
//    private and commercial purposes. Any commercial use is at the user’s 
//    own risk and responsibility.
//
// -------------------------------------------------------------------------
TYPE RobotCoordinateSystemParameters :
STRUCT
  /// Index of target tool
  /// • 0: Flange (default)
  /// • 1..254: Tool frames
  ToolNo : USINT;
  /// Index of target frame
  /// • 0: WCS (default)
  /// • 1..254: User frames
  FrameNo : USINT;  
END_STRUCT
END_TYPE

{attribute 'pack_mode' := '1'}
// ------------------------------------------------------------------------- 
//  SRCI Robot Library                                                
// ------------------------------------------------------------------------- 
//                                                                           
//  Object:      RspHeader                                       
//  Author:      Thorsten Brach                                                
//  Date:        2024-06-01
//
//  Description:                                              
//   
//                                                                           
//  Copyright: 
//    (C) 2024 Thorsten Brach. All rights reserved                                                                         
//                                                                           
//  Disclaimer:                                                                           
//    This project is provided without any guarantee and can be used for   
//    private and commercial purposes. Any commercial use is at the user’s 
//    own risk and responsibility.
//
// -------------------------------------------------------------------------
TYPE RspHeader :  
STRUCT
  /// Parameter Sequence, used to identify sets of CMD parameter - For more information see chapter 5.6.4
  ParSeq               : SequenceFlag;
  /// Actual state of the command - For more information and examples, see chapter 5.6.3.2
  State                : CmdMessageState;
  /// Severity of returned message according to .Table 5-47.
  AlarmMessageSeverity : Severity;
  /// Message code for error/warning/info identification reported during execution of command according to
  /// • Error: Table 7-1
  /// • Warning: Table 7-3
  /// • Info: Table 7-5
  AlarmMessageCode     : UINT;  
END_STRUCT
END_TYPE

{attribute 'pack_mode' := '1'} 
// ------------------------------------------------------------------------- 
//  SRCI Robot Library                                                
// ------------------------------------------------------------------------- 
//                                                                           
//  Object:      TimeStamp                                       
//  Author:      Thorsten Brach                                                
//  Date:        2024-06-01
//
//  Description:                                              
//   
//                                                                           
//  Copyright: 
//    (C) 2024 Thorsten Brach. All rights reserved                                                                         
//                                                                           
//  Disclaimer:                                                                           
//    This project is provided without any guarantee and can be used for   
//    private and commercial purposes. Any commercial use is at the user’s 
//    own risk and responsibility.
//
// -------------------------------------------------------------------------
TYPE TimeStamp :
STRUCT
  /// Date of the timestamp
  TsData : DATE;
  /// Time of the timestamp
  TsTime : TIME;
END_STRUCT
END_TYPE

{attribute 'pack_mode' := '1'} 
// ------------------------------------------------------------------------- 
//  SRCI Robot Library                                                
// ------------------------------------------------------------------------- 
//                                                                           
//  Object:      CyclicStateData                                       
//  Author:      Thorsten Brach                                                
//  Date:        2024-06-01
//
//  Description:                                              
//   
//                                                                           
//  Copyright: 
//    (C) 2024 Thorsten Brach. All rights reserved                                                                         
//                                                                           
//  Disclaimer:                                                                           
//    This project is provided without any guarantee and can be used for   
//    private and commercial purposes. Any commercial use is at the user’s 
//    own risk and responsibility.
//
// -------------------------------------------------------------------------
TYPE CyclicStateData :
STRUCT
  /// Combination of various RA related states.
  StatusWord : RaStatusWord;
  /// Actual override in percentage multiplied by 100 (see chapter 5.6.2 for more information about the percentage encoding)
  Override   : UINT;
END_STRUCT
END_TYPE

{attribute 'pack_mode' := '1'} 
// ------------------------------------------------------------------------- 
//  SRCI Robot Library                                                
// ------------------------------------------------------------------------- 
//                                                                           
//  Object:      FrameData                                       
//  Author:      Thorsten Brach                                                
//  Date:        2024-06-01
//
//  Description:                                              
//   
//                                                                           
//  Copyright: 
//    (C) 2024 Thorsten Brach. All rights reserved                                                                         
//                                                                           
//  Disclaimer:                                                                           
//    This project is provided without any guarantee and can be used for   
//    private and commercial purposes. Any commercial use is at the user’s 
//    own risk and responsibility.
//
// -------------------------------------------------------------------------
TYPE FrameData :
STRUCT
  /// Timestamp
  Timestamp      : DT;
  /// Frame to which the shifting and rotation is relative M
  ReferenceFrame : USINT;
  /// Origin of the coordinate system relative to the BCS/WCS/UCS 
  /// X value [mm]  
  X              : REAL := 0;
  /// Origin of the coordinate system relative to the BCS/WCS/UCS 
  /// Y value [mm]  
  Y              : REAL := 0;
  /// Origin of the coordinate system relative to the BCS/WCS/UCS 
  /// Z value [mm]  
  Z              : REAL := 0;
  /// Orientation of the coordinate system relative to the BCS/WCS/UCS
  /// Rx value [°]  
  Rx             : REAL := 0;
  /// Rx value [°]  
  Ry             : REAL := 0;
  /// Rx value [°]  
  Rz             : REAL := 0;  
END_STRUCT
END_TYPE

{attribute 'pack_mode' := '1'} 
// ------------------------------------------------------------------------- 
//  SRCI Robot Library                                                
// ------------------------------------------------------------------------- 
//                                                                           
//  Object:      LoadData                                       
//  Author:      Thorsten Brach                                                
//  Date:        2024-06-01
//
//  Description:                                              
//   
//                                                                           
//  Copyright: 
//    (C) 2024 Thorsten Brach. All rights reserved                                                                         
//                                                                           
//  Disclaimer:                                                                           
//    This project is provided without any guarantee and can be used for   
//    private and commercial purposes. Any commercial use is at the user’s 
//    own risk and responsibility.
//
// -------------------------------------------------------------------------
TYPE LoadData :
STRUCT
  /// Timestamp
  Timestamp : DT;
  /// Position of the center of gravity relative to the flange.
  /// X value [mm]  
  X         : REAL := 0;
  /// Position of the center of gravity relative to the flange.
  /// Y value [mm]  
  Y         : REAL := 0;
  /// Position of the center of gravity relative to the flange.
  /// Z value [mm]  
  Z         : REAL := 0;
  /// Orientation of the principal inertia axes relative to the flange. O
  /// Rx value [°]  
  Rx        : REAL := 0;
  /// Ry value [°]  
  Ry        : REAL := 0;
  /// Rz value [°]  
  Rz        : REAL := 0;
  /// The mass of the tool and workpiece being gripped. [kg]
  Mass      : REAL := 0;
  /// The moment of inertia of the load around the resulting inertia X-Axis [kg/m²]
  Ix        : REAL := 0;
  /// The moment of inertia of the load around the resulting inertia y-axis [kg/m²]
  Iy        : REAL := 0;
  /// The moment of inertia of the load around the resulting inertia z-axis [kg/m²]
  Iz        : REAL := 0;  
END_STRUCT
END_TYPE

{attribute 'pack_mode' := '1'} 
// ------------------------------------------------------------------------- 
//  SRCI Robot Library                                                
// ------------------------------------------------------------------------- 
//                                                                           
//  Object:      RobotSubProgramData                                       
//  Author:      Thorsten Brach                                                
//  Date:        2024-06-01
//
//  Description:                                              
//   
//                                                                           
//  Copyright: 
//    (C) 2024 Thorsten Brach. All rights reserved                                                                         
//                                                                           
//  Disclaimer:                                                                           
//    This project is provided without any guarantee and can be used for   
//    private and commercial purposes. Any commercial use is at the user’s 
//    own risk and responsibility.
//
// -------------------------------------------------------------------------
TYPE RobotSubProgramData :
STRUCT
  /// Sub program data
  Data : ARRAY [0..25] OF BYTE;
END_STRUCT
END_TYPE

{attribute 'pack_mode' := '1'} 
// ------------------------------------------------------------------------- 
//  SRCI Robot Library                                                
// ------------------------------------------------------------------------- 
//                                                                           
//  Object:      SplineData                                       
//  Author:      Thorsten Brach                                                
//  Date:        2024-06-01
//
//  Description:                                              
//   
//                                                                           
//  Copyright: 
//    (C) 2024 Thorsten Brach. All rights reserved                                                                         
//                                                                           
//  Disclaimer:                                                                           
//    This project is provided without any guarantee and can be used for   
//    private and commercial purposes. Any commercial use is at the user’s 
//    own risk and responsibility.
//
// -------------------------------------------------------------------------
TYPE SplineData :
STRUCT
    /// Absolute target coordinates in the selected coordinate system (see ToolNo and FrameNo).
    Position : RobotCartesianPosition;
    /// TCP velocity in % of nominal velocity.
    /// •  <0% : Use default velocity (default)
    /// •   0% : Use internal minimal velocity
    /// • 100% : Use maximal reference velocity
    /// • See chapter 5.5.7 Robot dynamics
    VelocityRate : REAL;    
    /// Acceleration for movement in % of nominal acceleration.
    /// •  <0% : Use default acceleration (default)
    /// •   0% : Use internal minimal acceleration
    /// • 100% : Use maximal reference acceleration
    /// • See chapter 5.5.7 Robot dynamics
    AccelerationRate : REAL;    
    /// Deceleration for movement in % of nominal deceleration.
    /// •  <0% : Use default deceleration (default)
    /// •   0% : Use internal minimal deceleration
    /// • 100% : Use maximal reference deceleration
    /// • See chapter 5.5.7 Robot dynamics
    DecelerationRate : REAL;    
    /// Jerk of the movement in % of nominal jerk.
    /// <0% o Use default jerk (default)
    /// 0% o Use internal minimal jerk
    /// 100% o Use maximal reference jerk
    /// See chapter 5.5.7 Robot dynamics
    JerkRate : REAL;
    /// Index of tool
    /// 0: Flange (default)
    /// 1..254: Tool frames
    ToolNo : USINT;    
    /// Index of frame
    /// 0: WCS (default)
    /// 1..254: User frames
    FrameNo : USINT;    
    /// [ms] Parameter is used if it is greater than 0 (default):
    /// Parameter defines the time for the movement to reach the target position
    /// Velocity input can be ignored
    /// Acceleration, Deceleration and jerk will be ignored
    /// Define two consecutive points with identical positions and specified Time to realize waiting time on spline.
    /// Error is sent by the RC, if the time cannot be kept.
    MoveTime : UINT;  
END_STRUCT
END_TYPE

{attribute 'pack_mode' := '1'} 
// ------------------------------------------------------------------------- 
//  SRCI Robot Library                                                
// ------------------------------------------------------------------------- 
//                                                                           
//  Object:      ToolData                                       
//  Author:      Thorsten Brach                                                
//  Date:        2024-06-01
//
//  Description:                                              
//   
//                                                                           
//  Copyright: 
//    (C) 2024 Thorsten Brach. All rights reserved                                                                         
//                                                                           
//  Disclaimer:                                                                           
//    This project is provided without any guarantee and can be used for   
//    private and commercial purposes. Any commercial use is at the user’s 
//    own risk and responsibility.
//
// -------------------------------------------------------------------------
TYPE ToolData :
STRUCT
  /// Timestamp
  Timestamp   : DT;
  /// Identification of physical tool Default: 0 
  ID          : USINT;
  /// True: Tool fixed False: Tool on flange 
  ExternalTCP : BOOL;
  /// Origin of the tool coordinate system relative to the flange coordinate system. 
  /// X value [mm]  
  X           : REAL;
  /// Origin of the tool coordinate system relative to the flange coordinate system. 
  /// Y value [mm]  
  Y           : REAL;
  /// Origin of the tool coordinate system relative to the flange coordinate system. 
  /// Z value [mm]  
  Z           : REAL;
  /// Orientation of the tool coordinate system relative to the flange coordinate system 
  /// RX value[°]
  Rx          : REAL;
  /// Orientation of the tool coordinate system relative to the flange coordinate system 
  /// RX value[°]
  Ry          : REAL;
  /// Orientation of the tool coordinate system relative to the flange coordinate system 
  /// RX value[°]
  Rz          : REAL;
  /// Index of the payload Information of tool and workpiece weight, center of gravity and inertia 
  LoadNo      : USINT;  
END_STRUCT
END_TYPE

{attribute 'pack_mode' := '1'} 
// ------------------------------------------------------------------------- 
//  SRCI Robot Library                                                
// ------------------------------------------------------------------------- 
//                                                                           
//  Object:      UserData                                       
//  Author:      Thorsten Brach                                                
//  Date:        2024-06-01
//
//  Description:                                              
//   
//                                                                           
//  Copyright: 
//    (C) 2024 Thorsten Brach. All rights reserved                                                                         
//                                                                           
//  Disclaimer:                                                                           
//    This project is provided without any guarantee and can be used for   
//    private and commercial purposes. Any commercial use is at the user’s 
//    own risk and responsibility.
//
// -------------------------------------------------------------------------
TYPE UserData :
STRUCT
  /// Set TRUE (default), to activate the synchronizationrelated comparison mechanism for tool data 
  EnableSyncTool                 : BOOL;
  /// Set TRUE (default), to activate the synchronizationrelated comparison mechanism for frame data
  EnableSyncFrame                : BOOL;
  /// Set TRUE (default), to activate the synchronizationrelated comparison mechanism for load data
  EnableSyncLoad                 : BOOL;
  /// Set TRUE (default), to activate the synchronizationrelated comparison mechanism for work area data
  EnableSyncWorkArea             : BOOL;
  /// Set TRUE (default), to activate the synchronizationrelated comparison mechanism for software limits
  EnableSyncSWLimits             : BOOL;
  /// Set TRUE (default), to activate the synchronizationrelated comparison mechanism for default dynamics
  EnableSyncDefaultDynamics      : BOOL;
  /// Set TRUE (default), to activate the synchronizationrelated comparison mechanism for reference dynamics
  EnableSyncReferenceDynamics    : BOOL;
  /// Set TRUE to define two sequences in one Telegram.
  ActivateTwoSequences           : BOOL;
  /// Define direction of synchronization for tool data according to Table 6-4
  SyncModeTool                   : SINT;
  /// Define direction of synchronization for frame data according to Table 6-4  
  SyncModeFrame                  : SINT;
  /// Define direction of synchronization for load data according to Table 6-4
  SyncModeLoad                   : SINT;
  /// Define direction of synchronization for work area data according to Table 6-4
  SyncModeWorkAreas              : SINT;
  /// Define direction of synchronization for software limits according to Table 6-4
  SyncModeSWLimits               : SINT;
  /// Define direction of synchronization for default dynamics according to Table 6-4
  SyncModeDefaultDynamics        : SINT;
  /// Define direction of synchronization for reference dynamics according to Table 6-4
  SyncModeReferenceDynamics      : SINT;
  /// Defines waiting time [ms] of RC between receiving a first move command when motion queue is empty and starting the first movement. See also chapter 5.6.8.
  DelayTime                      : UINT; 
  /// Define number of points required to calculate the blending. See also chapter 5.6.8
  WaitForNrOfCmd                 : UINT;
  ///Defines blending behavior for single move commands
  /// • 0 (default): Move to end position :
  ///     Robot moves exactly the target position independently of the selected "BlendingMode"
  /// 
  /// • 1: Wait at blending parameter : 
  ///      Robot stops its movement when the specified blending parameter is reached
  WaitAtBlendingZone             : BOOL;
  /// Allow a sequence switch from primary to secondary while a subprogram called via CallSubprogram (6.5.18) in the sequence is in progress
  AllowSecSeqWhileSubprogram     : BOOL;
  /// Allows blending when CallSubprogram is called in sequence and removed afterwards.
  /// For more information see chapter 6.5.21.
  /// • 0 (default): Dynamic blending is prevented
  /// • 1: Dynamic blending is allowed
  AllowDynamicBlending           : BOOL;
  /// Maximum allowed time [ms] between incrementation of LifeSign before communication error.
  /// • <10 ms: Invalid
  /// • 50 ms: default
  /// See also chapter 5.6.6.2.
  LifeSignTimeOut                : UINT;
  /// Specifies system reaction in case inconsistency of synchronization data is detected according to Table 6-81. For more information refer to chapter 5.6.7.2
  SyncReaction                   : USINT;
  /// Defines a delay time [ms] between detecting an inconsistency of configuration data between server and client an executing the defined SyncReaction.
  /// Always positive.
  /// • Default: 0 ms
  SyncDelay                      : UINT;
  /// Defines up to which level of severity messages will be logged in the RC's server log
  LogLevel                       : LogLevel;
  /// Defines up to which level of severity messages will be transmitted to the PLC’s message buffer
  MessageLevel                   : MessageLevel;
  /// Version of client implementation in format (X.X.X)
  PLCLibraryVersion              : VersionStruct;
  /// RC manufacturer name 
  RCManufacturer                 : STRING(20); 
  /// RC part number 
  RCOrderID                      : STRING(20); 
  /// RC serial number 
  RCSerialNumber                 : STRING(16); 
  /// RA serial number 
  RASerialNumber                 : STRING(16); 
  /// Robot firmware version in manufacturer-specific format 
  RCFirmwareVersion              : STRING(12); 
  /// Version of server implementation in format (X.X.X) 
  RCInterpreterVersion           : VersionStruct;
  /// Version of SRCI specification on which server implementation is based in format (X.X.X)  
  RCSRCIVersion                  : VersionStruct;
  /// TRUE  = Axis used in Robot, FALSE = Axis NOT used. See Table 6-13 for bit assignment.
  AxisJointUsed                  : BYTE;
  /// TRUE = Axis used by Robot, FALSE = Axis NOT used. See Table 6-13 for bit assignment.
  AxisExternalUsed               : BYTE;
  /// TRUE = mm, FALSE = °. See Table 6-13 for bit assignment.
  AxisJointUnit                  : BYTE;
  /// TRUE = mm, FALSE = °. See Table 6-13 for bit assignment.
  AxisExternalUnit               : BYTE;
  /// Interface is initialized and ready to process commands.
  Initialized                    : BOOL;
  /// All synchronization-related configuration data between client and server is synchronized.
  Synchronized                   : BOOL;
  /// ToolData synchronization is activated.
  ToolDataSynchronizing          : BOOL;
  /// FrameData synchronization is activated.
  FrameDataSynchronizing         : BOOL;
  /// LoadData synchronization is activated.
  LoadDataSynchronizing          : BOOL;
  /// WorkAreaData synchronization is activated.
  WorkAreaDataSynchronizing      : BOOL;
  /// SWLimits synchronization is activated.
  SWLimitsSynchronizing          : BOOL;
  /// DefaultDynamics synchronization is activated.
  DefaultDynamicsSynchronizing   : BOOL;
  /// ReferenceDynamics synchronization is activated.
  ReferenceDynamicsSynchronizing : BOOL;
  /// TRUE, when robot’s axes values change due to physical movement of axes. Can only be TRUE in sequence state "Executing". Default: FALSE 
  IsMoving                       : BOOL;
  /// TRUE, when move commands buffered by the primary sequence are currently not processed. Default: FALSE 
  PrimarySequencePaused          : BOOL;
  /// TRUE, when robot is moving in the primary sequence. FALSE, when robot leaves its position by other means than move commands in the primary sequence. Default: FALSE
  InPrimaryPos                   : BOOL;
  /// TRUE, when secondary sequence is active. Default: FALSE
  SecondarySequenceActive        : BOOL;
  /// Shows that an error acknowledgement by the client is necessary. Default: FALSE
  ErrorPending                   : BOOL;
  /// TRUE, when RC is restarting. Default: FALSE
  RestartInProgress              : BOOL;
  /// Signals that a brake test is required in the defined monitoring time (see chapter 6.5.27).
  BrakeTestRequired              : BOOL;
  /// RA power state. Default: FALSE
  Enabled                        : BOOL;
  /// TRUE, while RA sequence states returns Idle. Default: FALSE
  Idle                           : BOOL;
  /// TRUE, while RA sequence states returns Executing. Default: FALSE
  Executing                      : BOOL;
  /// TRUE, while RA sequence states returns Interrupted. Default: FALSE
  Interrupted                    : BOOL;
  /// TRUE, when robot is currently blending between to move commands. Can only be TRUE in sequence state "Executing". Default: FALSE
  IsBlending                     : BOOL;  
  /// Operation Mode (see chapter 5.5.1)
  OperationMode                  : USINT;
  /// PathAccuracyMode is active (see chapter 6.5.22) 
  PathAccuracyMode               : BOOL;
  /// AvoidSingularity is active (see chapter 6.5.23) 
  AvoidSingularity               : BOOL;
  /// TRUE, while CollisionDetection is enabled (see chapter 6.5.35) Default: FALSE 
  CollisionDetectionEnabled      : BOOL;
  /// TRUE, when a collision was detected while CollisionDetection is enabled (see chapter 6.5.35) Default: FALSE 
  CollisionDetected              : BOOL;
  /// TRUE, when the RC requests a restart of the RC induced through the functions "WriteRobotSWLimits" (chapter 6.2.16) or "WriteSystemVariable" (chapter 6.5.8) Default: FALSE 
  RestartRequested               : BOOL;
  /// Actual override
  ActualOverride                 : UINT;
  /// StepMode is active and set to ExactStop (see chapter 6.1.3) 
  StepModeExactStopActive        : BOOL;
  /// StepMode is active and set to Blending (see chapter 6.1.3) 
  StepModeBlendingActive         : BOOL;
  /// Cyclic dynamics status bit Accelerating is supported by RC (see chapter 5.5.3.2) 
  AcceleratingSupported          : BOOL;
  /// TRUE, when the robot is currently accelerating Default: FALSE 
  Accelerating                   : BOOL;
  /// Cyclic dynamics status bit Decelerating is supported by RC (see chapter 5.5.3.2) 
  DeceleratingSupported          : BOOL;
  /// TRUE, when the robot is currently decelerating Default: FALSE 
  Decelerating                   : BOOL;
  /// Cyclic dynamics status bit ConstantVelocity is supported by RC (see chapter 5.5.3.2) 
  ConstantVelocitySupported      : BOOL;
  /// TRUE, while the robot velocity is constant Default: FALSE 
  ConstantVelocity               : BOOL;
  /// TRUE, while the CartesianPosition is returned cyclically 
  ReadingCartesianPosition       : BOOL;
  /// TRUE, while the ExtCartesianPosition is returned cyclically 
  ReadingExtCartesianPosition    : BOOL;
  /// TRUE, while the JointPosition is returned cyclically 
  ReadingJointPosition           : BOOL;
  /// TRUE, while the ExtJointPosition is returned cyclically 
  ReadingExtJointPosition        : BOOL;
  /// Cyclically returned, absolute coordinates of current position in selected coordinate systems (see input parameters ToolNo and FrameNo of function ReadActualPositionCyclic 6.1.6)
  CartesianPosition              : RobotCartesianPositionShort;
  /// Cyclically returned, absolute cartesian position of the external axes of the robot in selected coordinate systems (see input parameters ToolNo and FrameNo of function ReadActualPositionCyclic 6.1.6)
  ExtCartesianPosition           : RobotCartesianPositionExt;  
  /// Cyclically returned, absolute position of the robot in Joint position
  JointPosition                  : RobotJointPositionShort;
  /// Cyclically returned, absolute joint position of the external axes of the robot
  ExtJointPosition               : RobotJointPositionExt;
  /// TRUE: Function is supported by RC
  /// FALSE: Function is not supported by RC
  /// See Table 6-14 for bit assignment.
  RCSupportedFunctions           : RCSupportedFunctions;
END_STRUCT
END_TYPE

